ABB RobotStudio station: ProyectoC2_Bohorquez_Parga_Torres.rspag

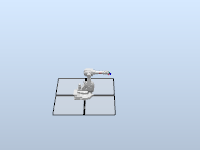
--- station ---
Station ProyectoC2_Bohorquez_Parga_Torres (saved by RobotStudio 20.4.9280.0)
Controller IRB1600_10_120
  mechanical unit ROB_1: IRB1600_10_120__01, 6 joints, base frame (0, 0, 0) mm
Layout (positions relative to the parent item):
  - IRB1600_10_120__01 [mechanism, from Robots\IRB1600_10_120_G_01.rslib] at (0, 0, 0) mm; joint values [0, 0, 0, 0, 0.5236, 0] (rad or m)

--- Backups/IRB1600_10_120/RAPID/TASK1/PROGMOD/Module1.mod ---
MODULE Module1
    !***********************************************************
    !
    ! Module:  Module1
    !
    ! Description:
    !   <Insert description here>
    !
    ! Author: Camilo
    !
    ! Version: 1.0
    !
    !***********************************************************


    !***********************************************************
    !
    ! Procedure main
    !
    !   This is the entry point of your program
    !
    !***********************************************************
    PROC main()
        !Add your code here
    ENDPROC
ENDMODULE
